PROGRAM MAIN
VAR
	Event_Buffer : EventBuffer;
	
	addEvent : BOOL;
	addEvent2 :BOOL;
	stEventToAdd :ST_Event;
	bEventToAddError : BOOL;
	
	
	ReadAndRemoved_Event : BOOL;
    ReadAndRemoved_Event2 : BOOL;
	stLastReadEvent: ST_Event;
	stLastReadEvent2: ST_Event;
	bReadAndRemoveEventError : BOOL;
END_VAR


IF AddEvent THEN 
	Event_Buffer.AddEvent(st_Event:= stEventToAdd, bError =>	bEventToAddError );
	addEvent := FALSE;
END_IF

IF ReadAndRemoved_Event THEN 
	
	Event_Buffer.ReadAndRemoveEvent(stEvent => stLastReadEvent, bError =>	bReadAndRemoveEventError );
	ReadAndRemoved_Event := FALSE;
END_IF

END_PROGRAM

(* stored: Version 1.1.0.1, ProductVersion 3.1.4024.9
   POU MAIN: Id {c3eb43f8-e5e6-41e3-a9bd-75fbe1d2c349}, SpecialFunc None *)
